FUNCTION_BLOCK FB_AxisHandautomatic_1
VAR_INPUT
    Notmoing:BOOL;//主轴停止中
	Run:BOOL;//自动
	i:INT;
	j: INT;
	Reset:BOOL;//手自动对比复位
END_VAR

VAR_OUTPUT
error :BOOL ;
END_VAR

VAR
	step:INT ;
	rRun : R_TRIG;
	fRun: F_TRIG;

	Pause_CMD:ARRAY[1..185] OF LREAL ; //手自动对比位置
	Handautomark:BOOL;//手自动对比标志
	K: INT;
	K1: INT;

END_VAR

VAR_IN_OUT

END_VAR




rRun(CLK:= Run , Q=> );
fRun(CLK:= Run , Q=> );


		IF fRun.Q THEN
			step:=100; 
		END_IF
		
	CASE step OF	
		100:
		   IF Notmoing THEN
			 step:=110;  
		   END_IF
	    110:    
	        Handautomark:=TRUE;
			FOR K:=i TO ((i+j)-1) DO 
				IF   K<>166 AND K<>167 AND K<>168  THEN
			          Pause_CMD[K]:=arrAxisCtrl[K].Status.fActPos;
				END_IF	  
			END_FOR
			Pause_CMD[166]:=arrAxisCtrlV2[166].Status.fActPos;
			Pause_CMD[167]:=arrAxisCtrlV2[167].Status.fActPos;
			Pause_CMD[168]:=arrAxisCtrlV2[168].Status.fActPos;
			
	        step:=120;    
	END_CASE
		

	   IF rRun.Q AND Handautomark THEN
				FOR K:=i TO ((i+j)-1) DO 
						IF  ABS(Pause_CMD[K]-arrAxisCtrl[K].Status.fActPos)>=0.2 AND K<>166 AND K<>167 AND K<>168  THEN
						Axis_error[k]:=TRUE;
						END_IF
			
						IF  ABS(Pause_CMD[166]-arrAxisCtrlV2[166].Status.fActPos)>0.2  THEN
						Axis_error[166]:=TRUE;
						END_IF

						IF  ABS(Pause_CMD[167]-arrAxisCtrlV2[167].Status.fActPos)>0.2  THEN
						Axis_error[167]:=TRUE;
						END_IF

						IF  ABS(Pause_CMD[168]-arrAxisCtrlV2[168].Status.fActPos)>0.2  THEN
						Axis_error[168]:=TRUE;
						END_IF
			
						IF Axis_error[k]   THEN
							error:=TRUE;
						END_IF
				END_FOR
				    Handautomark:=FALSE;
		END_IF
		
		IF stSysState.btnReset OR  stSysState.hmiReset  THEN
			   error:=FALSE;
			   FOR K1:=1 TO 185 DO 
				       Axis_error [K1]:=FALSE;
			   END_FOR
		END_IF
		
		IF Reset THEN
			 Handautomark:=FALSE;
		END_IF

END_FUNCTION_BLOCK

(* stored: Version 1.1.0.1, ProductVersion 3.1.4024.9
   POU FB_AxisHandautomatic_1: Id {6e9e61b9-0e80-48e4-b7a9-5e2a92667f7f}, SpecialFunc None *)
